{attribute 'qualified_only'}
VAR_GLOBAL PERSISTENT
	b_recipe_backup	:BOOL;
	
	b_recipe_bool_change :BOOL; //sygnał, że ktoś zmienił parametr bool
	b_recipe_real_change :BOOL; //sygnał, że ktoś zmienił parametr inny
	i_recipe_change :INT;
	lr_recipe_change :LREAL; //stara wartość w polu lr_param
	
	b_recipe_change_1 :BOOL;
	i_recipe_change_1 :INT;
	lr_recipe_change_1 :LREAL; //nowa wartość w polu lr_param
	
	s_recipe_change    :WSTRING(200); //kto zmienił parametr
	s_recipe_change_1  :WSTRING(200); //jaki parametr
	s_recipe_change_2  :WSTRING(200); //zmienna receptury
	s_recipe_change_3  :WSTRING(300); //zmienna do kontrolki
	b_old_recipe_param :BOOL; //stara wartość parametru b_param
	b_new_recipe_param :BOOL; //nowa wartość parametru b_param
	

	
	s_recipe_value :STRING;
	ArRecipeChanges: ARRAY [0..500] OF st_recipe_changes;	
	s_recipe_name :WSTRING(200); //nazwa receptury
	s_recupe_change_4 :WSTRING(200);
	b_recipe_changes_clear :BOOL:=FALSE;
END_VAR

(* stored: Version 1.1.0.1, ProductVersion 3.1.4026.13, FileIdentifier 5bfa7c22e4851d2473f642d500a1d403a28483d8, FileSignature 5a9708b2f5f989a5712215020cbe0ef22806f16959ccc9c7f2d267e07b6a0869a30e3efa4bf71b7e282a6dee8a9dcc2c5bd32b8906eff0b43ec8df7279ef9311b927ef5bb3f04e941797c3c5363f257039834b9ff8181c3a3fc8e5422512821efc395fd5dab05bb54186a540fbe82a07da4aa98d0a893b20e02c7e5837af3a104a22dda2e9bc8306a52a9c19a3be94c85d0326116271a36483a055efa0c3386fe25f58342418f1e627a70d464b0f4dbb4797acda7b70d45c2fae344e254ff1cf7fdb7988a22ae8ae9eda77627dac622e98c6c1c2b4492bb25564651217aa8c860526e18b7bfceeaaf52e7af25f9ce65c8f2d49b4c664689a37da8e13821bb76b
   GVL GVL_Recipe: Id {52970311-9775-474a-a82b-0858d99ac1aa} *)
